// TIA Portal V18 export
// export: Created 2026-06-08T14:19:27.3294129Z, ExportSetting WithDefaults, DisplayName Totally Integrated Automation Portal, DisplayVersion V18, DisplayName TIA Portal Openness, DisplayVersion V18, DisplayName TIA Portal Version Control Interface, DisplayVersion V18, DisplayName STEP 7 Professional, DisplayVersion V18, DisplayName STEP 7 Safety, DisplayVersion V18, DisplayName WinCC Professional, DisplayVersion V18
ORGANIZATION_BLOCK "Main"   // OB1, LAD, ProgramCycle
TITLE = "Main Program Sweep (Cycle)"
{ S7_Optimized_Access := 'TRUE' }
VERSION : 0.1
// stored: AutoNumber true, IsIECCheckEnabled false, SetENOAutomatically false
   VAR_INPUT
      Initial_Call : Bool;   // Initial call of this OB
      Remanence : Bool;   // =True, if remanent data are available
   END_VAR
BEGIN

REGION Network 1: PLC1 - Gọi logic khởi tạo recipe mặc định PLC1
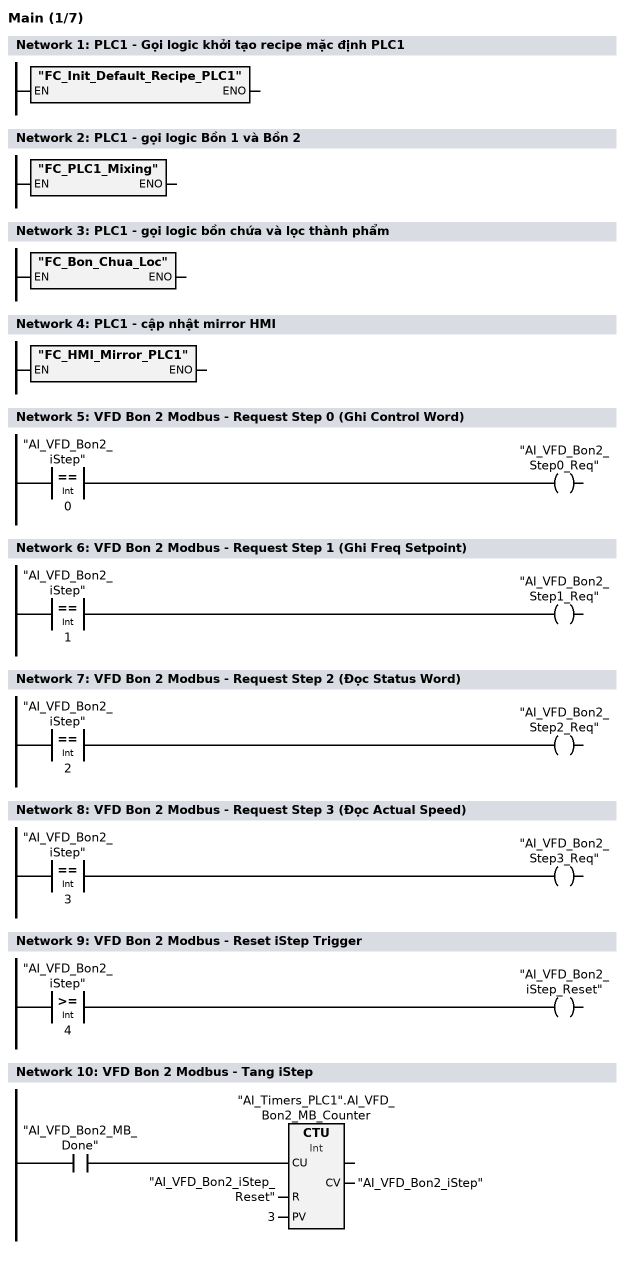
   RUNG wire#powerrail
      "FC_Init_Default_Recipe_PLC1"()
   END_RUNG
   // the same network as SCL:
   "FC_Init_Default_Recipe_PLC1"();
END_REGION

REGION Network 2: PLC1 - gọi logic Bồn 1 và Bồn 2
   RUNG wire#powerrail
      "FC_PLC1_Mixing"()
   END_RUNG
   // the same network as SCL:
   "FC_PLC1_Mixing"();
END_REGION

REGION Network 3: PLC1 - gọi logic bồn chứa và lọc thành phẩm
   RUNG wire#powerrail
      "FC_Bon_Chua_Loc"()
   END_RUNG
   // the same network as SCL:
   "FC_Bon_Chua_Loc"();
END_REGION

REGION Network 4: PLC1 - cập nhật mirror HMI
   RUNG wire#powerrail
      "FC_HMI_Mirror_PLC1"()
   END_RUNG
   // the same network as SCL:
   "FC_HMI_Mirror_PLC1"();
END_REGION

REGION Network 5: VFD Bon 2 Modbus - Request Step 0 (Ghi Control Word)
   RUNG wire#powerrail
      { S7_Templates := "SrcType := Int" } EQ_Contact(in1 := "AI_VFD_Bon2_iStep", in2 := 0)
      Coil( "AI_VFD_Bon2_Step0_Req" )
   END_RUNG
   // the same network as SCL:
   "AI_VFD_Bon2_Step0_Req" := "AI_VFD_Bon2_iStep" = 0;
END_REGION

REGION Network 6: VFD Bon 2 Modbus - Request Step 1 (Ghi Freq Setpoint)
   RUNG wire#powerrail
      { S7_Templates := "SrcType := Int" } EQ_Contact(in1 := "AI_VFD_Bon2_iStep", in2 := 1)
      Coil( "AI_VFD_Bon2_Step1_Req" )
   END_RUNG
   // the same network as SCL:
   "AI_VFD_Bon2_Step1_Req" := "AI_VFD_Bon2_iStep" = 1;
END_REGION

REGION Network 7: VFD Bon 2 Modbus - Request Step 2 (Đọc Status Word)
   RUNG wire#powerrail
      { S7_Templates := "SrcType := Int" } EQ_Contact(in1 := "AI_VFD_Bon2_iStep", in2 := 2)
      Coil( "AI_VFD_Bon2_Step2_Req" )
   END_RUNG
   // the same network as SCL:
   "AI_VFD_Bon2_Step2_Req" := "AI_VFD_Bon2_iStep" = 2;
END_REGION

REGION Network 8: VFD Bon 2 Modbus - Request Step 3 (Đọc Actual Speed)
   RUNG wire#powerrail
      { S7_Templates := "SrcType := Int" } EQ_Contact(in1 := "AI_VFD_Bon2_iStep", in2 := 3)
      Coil( "AI_VFD_Bon2_Step3_Req" )
   END_RUNG
   // the same network as SCL:
   "AI_VFD_Bon2_Step3_Req" := "AI_VFD_Bon2_iStep" = 3;
END_REGION

REGION Network 9: VFD Bon 2 Modbus - Reset iStep Trigger
   RUNG wire#powerrail
      { S7_Templates := "SrcType := Int" } GE_Contact(in1 := "AI_VFD_Bon2_iStep", in2 := 4)
      Coil( "AI_VFD_Bon2_iStep_Reset" )
   END_RUNG
   // the same network as SCL:
   "AI_VFD_Bon2_iStep_Reset" := "AI_VFD_Bon2_iStep" >= 4;
END_REGION

REGION Network 10: VFD Bon 2 Modbus - Tang iStep
   RUNG wire#powerrail
      Contact( "AI_VFD_Bon2_MB_Done" )
      { S7_Templates := "value_type := Int" } "AI_Timers_PLC1".AI_VFD_Bon2_MB_Counter.CTU(r := "AI_VFD_Bon2_iStep_Reset", pv := 3, cv => "AI_VFD_Bon2_iStep")
   END_RUNG
   // the same network as SCL:
   "AI_Timers_PLC1".AI_VFD_Bon2_MB_Counter.CTU(CU := "AI_VFD_Bon2_MB_Done",
                           R := "AI_VFD_Bon2_iStep_Reset",
                           PV := 3,
                           CV => "AI_VFD_Bon2_iStep");
END_REGION

REGION Network 11: VFD Bon 2 Modbus - Khoi tao RS-485
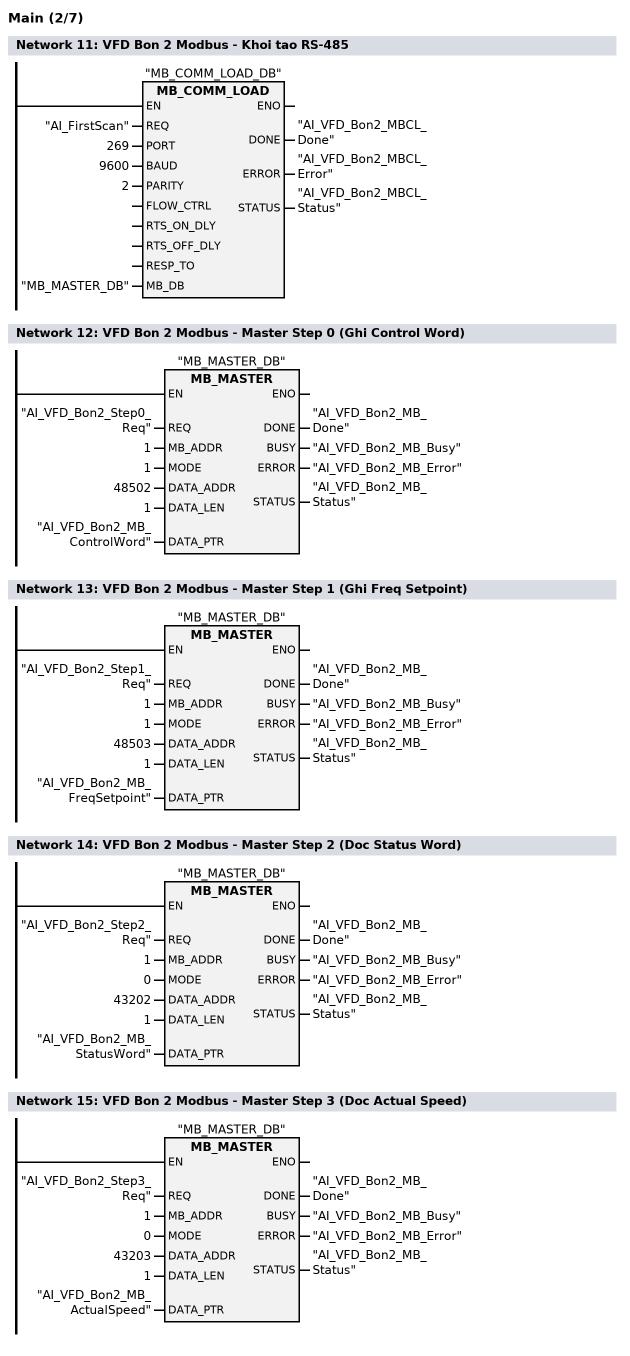
   RUNG wire#powerrail
      "MB_COMM_LOAD_DB".MB_COMM_LOAD(REQ := "AI_FirstScan", PORT := 269, BAUD := 9600, PARITY := 2, FLOW_CTRL :=, RTS_ON_DLY :=, RTS_OFF_DLY :=, RESP_TO :=, MB_DB := "MB_MASTER_DB", DONE => "AI_VFD_Bon2_MBCL_Done", ERROR => "AI_VFD_Bon2_MBCL_Error", STATUS => "AI_VFD_Bon2_MBCL_Status")
   END_RUNG
   // the same network as SCL:
   "MB_COMM_LOAD_DB"(REQ := "AI_FirstScan",   // MB_COMM_LOAD
                     PORT := 269,
                     BAUD := 9600,
                     PARITY := 2,
                     MB_DB := "MB_MASTER_DB",
                     DONE => "AI_VFD_Bon2_MBCL_Done",
                     ERROR => "AI_VFD_Bon2_MBCL_Error",
                     STATUS => "AI_VFD_Bon2_MBCL_Status");
END_REGION

REGION Network 12: VFD Bon 2 Modbus - Master Step 0 (Ghi Control Word)
   RUNG wire#powerrail
      "MB_MASTER_DB".MB_MASTER(REQ := "AI_VFD_Bon2_Step0_Req", MB_ADDR := 1, MODE := 1, DATA_ADDR := 48502, DATA_LEN := 1, DATA_PTR := "AI_VFD_Bon2_MB_ControlWord", DONE => "AI_VFD_Bon2_MB_Done", BUSY => "AI_VFD_Bon2_MB_Busy", ERROR => "AI_VFD_Bon2_MB_Error", STATUS => "AI_VFD_Bon2_MB_Status")
   END_RUNG
   // the same network as SCL:
   "MB_MASTER_DB"(REQ := "AI_VFD_Bon2_Step0_Req",   // MB_MASTER
                  MB_ADDR := 1,
                  MODE := 1,
                  DATA_ADDR := 48502,
                  DATA_LEN := 1,
                  DATA_PTR := "AI_VFD_Bon2_MB_ControlWord",
                  DONE => "AI_VFD_Bon2_MB_Done",
                  BUSY => "AI_VFD_Bon2_MB_Busy",
                  ERROR => "AI_VFD_Bon2_MB_Error",
                  STATUS => "AI_VFD_Bon2_MB_Status");
END_REGION

REGION Network 13: VFD Bon 2 Modbus - Master Step 1 (Ghi Freq Setpoint)
   RUNG wire#powerrail
      "MB_MASTER_DB".MB_MASTER(REQ := "AI_VFD_Bon2_Step1_Req", MB_ADDR := 1, MODE := 1, DATA_ADDR := 48503, DATA_LEN := 1, DATA_PTR := "AI_VFD_Bon2_MB_FreqSetpoint", DONE => "AI_VFD_Bon2_MB_Done", BUSY => "AI_VFD_Bon2_MB_Busy", ERROR => "AI_VFD_Bon2_MB_Error", STATUS => "AI_VFD_Bon2_MB_Status")
   END_RUNG
   // the same network as SCL:
   "MB_MASTER_DB"(REQ := "AI_VFD_Bon2_Step1_Req",   // MB_MASTER
                  MB_ADDR := 1,
                  MODE := 1,
                  DATA_ADDR := 48503,
                  DATA_LEN := 1,
                  DATA_PTR := "AI_VFD_Bon2_MB_FreqSetpoint",
                  DONE => "AI_VFD_Bon2_MB_Done",
                  BUSY => "AI_VFD_Bon2_MB_Busy",
                  ERROR => "AI_VFD_Bon2_MB_Error",
                  STATUS => "AI_VFD_Bon2_MB_Status");
END_REGION

REGION Network 14: VFD Bon 2 Modbus - Master Step 2 (Doc Status Word)
   RUNG wire#powerrail
      "MB_MASTER_DB".MB_MASTER(REQ := "AI_VFD_Bon2_Step2_Req", MB_ADDR := 1, MODE := 0, DATA_ADDR := 43202, DATA_LEN := 1, DATA_PTR := "AI_VFD_Bon2_MB_StatusWord", DONE => "AI_VFD_Bon2_MB_Done", BUSY => "AI_VFD_Bon2_MB_Busy", ERROR => "AI_VFD_Bon2_MB_Error", STATUS => "AI_VFD_Bon2_MB_Status")
   END_RUNG
   // the same network as SCL:
   "MB_MASTER_DB"(REQ := "AI_VFD_Bon2_Step2_Req",   // MB_MASTER
                  MB_ADDR := 1,
                  MODE := 0,
                  DATA_ADDR := 43202,
                  DATA_LEN := 1,
                  DATA_PTR := "AI_VFD_Bon2_MB_StatusWord",
                  DONE => "AI_VFD_Bon2_MB_Done",
                  BUSY => "AI_VFD_Bon2_MB_Busy",
                  ERROR => "AI_VFD_Bon2_MB_Error",
                  STATUS => "AI_VFD_Bon2_MB_Status");
END_REGION

REGION Network 15: VFD Bon 2 Modbus - Master Step 3 (Doc Actual Speed)
   RUNG wire#powerrail
      "MB_MASTER_DB".MB_MASTER(REQ := "AI_VFD_Bon2_Step3_Req", MB_ADDR := 1, MODE := 0, DATA_ADDR := 43203, DATA_LEN := 1, DATA_PTR := "AI_VFD_Bon2_MB_ActualSpeed", DONE => "AI_VFD_Bon2_MB_Done", BUSY => "AI_VFD_Bon2_MB_Busy", ERROR => "AI_VFD_Bon2_MB_Error", STATUS => "AI_VFD_Bon2_MB_Status")
   END_RUNG
   // the same network as SCL:
   "MB_MASTER_DB"(REQ := "AI_VFD_Bon2_Step3_Req",   // MB_MASTER
                  MB_ADDR := 1,
                  MODE := 0,
                  DATA_ADDR := 43203,
                  DATA_LEN := 1,
                  DATA_PTR := "AI_VFD_Bon2_MB_ActualSpeed",
                  DONE => "AI_VFD_Bon2_MB_Done",
                  BUSY => "AI_VFD_Bon2_MB_Busy",
                  ERROR => "AI_VFD_Bon2_MB_Error",
                  STATUS => "AI_VFD_Bon2_MB_Status");
END_REGION

REGION Network 16: Handshake Client - Reset Any Cmd Edge Flag
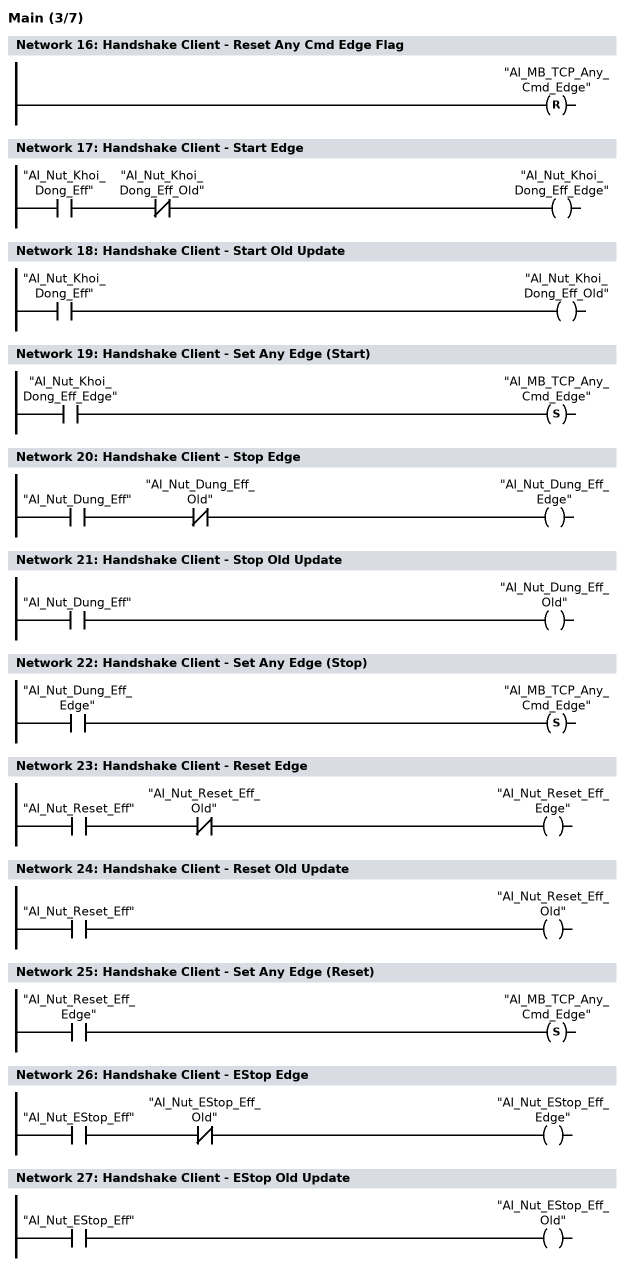
   RUNG wire#powerrail
      R_Coil( "AI_MB_TCP_Any_Cmd_Edge" )
   END_RUNG
   // the same network as SCL:
   "AI_MB_TCP_Any_Cmd_Edge" := FALSE;
END_REGION

REGION Network 17: Handshake Client - Start Edge
   RUNG wire#powerrail
      Contact( "AI_Nut_Khoi_Dong_Eff" )
      I_Contact( "AI_Nut_Khoi_Dong_Eff_Old" )
      Coil( "AI_Nut_Khoi_Dong_Eff_Edge" )
   END_RUNG
   // the same network as SCL:
   "AI_Nut_Khoi_Dong_Eff_Edge" := "AI_Nut_Khoi_Dong_Eff" AND NOT "AI_Nut_Khoi_Dong_Eff_Old";
END_REGION

REGION Network 18: Handshake Client - Start Old Update
   RUNG wire#powerrail
      Contact( "AI_Nut_Khoi_Dong_Eff" )
      Coil( "AI_Nut_Khoi_Dong_Eff_Old" )
   END_RUNG
   // the same network as SCL:
   "AI_Nut_Khoi_Dong_Eff_Old" := "AI_Nut_Khoi_Dong_Eff";
END_REGION

REGION Network 19: Handshake Client - Set Any Edge (Start)
   RUNG wire#powerrail
      Contact( "AI_Nut_Khoi_Dong_Eff_Edge" )
      S_Coil( "AI_MB_TCP_Any_Cmd_Edge" )
   END_RUNG
   // the same network as SCL:
   IF "AI_Nut_Khoi_Dong_Eff_Edge" THEN "AI_MB_TCP_Any_Cmd_Edge" := TRUE; END_IF;
END_REGION

REGION Network 20: Handshake Client - Stop Edge
   RUNG wire#powerrail
      Contact( "AI_Nut_Dung_Eff" )
      I_Contact( "AI_Nut_Dung_Eff_Old" )
      Coil( "AI_Nut_Dung_Eff_Edge" )
   END_RUNG
   // the same network as SCL:
   "AI_Nut_Dung_Eff_Edge" := "AI_Nut_Dung_Eff" AND NOT "AI_Nut_Dung_Eff_Old";
END_REGION

REGION Network 21: Handshake Client - Stop Old Update
   RUNG wire#powerrail
      Contact( "AI_Nut_Dung_Eff" )
      Coil( "AI_Nut_Dung_Eff_Old" )
   END_RUNG
   // the same network as SCL:
   "AI_Nut_Dung_Eff_Old" := "AI_Nut_Dung_Eff";
END_REGION

REGION Network 22: Handshake Client - Set Any Edge (Stop)
   RUNG wire#powerrail
      Contact( "AI_Nut_Dung_Eff_Edge" )
      S_Coil( "AI_MB_TCP_Any_Cmd_Edge" )
   END_RUNG
   // the same network as SCL:
   IF "AI_Nut_Dung_Eff_Edge" THEN "AI_MB_TCP_Any_Cmd_Edge" := TRUE; END_IF;
END_REGION

REGION Network 23: Handshake Client - Reset Edge
   RUNG wire#powerrail
      Contact( "AI_Nut_Reset_Eff" )
      I_Contact( "AI_Nut_Reset_Eff_Old" )
      Coil( "AI_Nut_Reset_Eff_Edge" )
   END_RUNG
   // the same network as SCL:
   "AI_Nut_Reset_Eff_Edge" := "AI_Nut_Reset_Eff" AND NOT "AI_Nut_Reset_Eff_Old";
END_REGION

REGION Network 24: Handshake Client - Reset Old Update
   RUNG wire#powerrail
      Contact( "AI_Nut_Reset_Eff" )
      Coil( "AI_Nut_Reset_Eff_Old" )
   END_RUNG
   // the same network as SCL:
   "AI_Nut_Reset_Eff_Old" := "AI_Nut_Reset_Eff";
END_REGION

REGION Network 25: Handshake Client - Set Any Edge (Reset)
   RUNG wire#powerrail
      Contact( "AI_Nut_Reset_Eff_Edge" )
      S_Coil( "AI_MB_TCP_Any_Cmd_Edge" )
   END_RUNG
   // the same network as SCL:
   IF "AI_Nut_Reset_Eff_Edge" THEN "AI_MB_TCP_Any_Cmd_Edge" := TRUE; END_IF;
END_REGION

REGION Network 26: Handshake Client - EStop Edge
   RUNG wire#powerrail
      Contact( "AI_Nut_EStop_Eff" )
      I_Contact( "AI_Nut_EStop_Eff_Old" )
      Coil( "AI_Nut_EStop_Eff_Edge" )
   END_RUNG
   // the same network as SCL:
   "AI_Nut_EStop_Eff_Edge" := "AI_Nut_EStop_Eff" AND NOT "AI_Nut_EStop_Eff_Old";
END_REGION

REGION Network 27: Handshake Client - EStop Old Update
   RUNG wire#powerrail
      Contact( "AI_Nut_EStop_Eff" )
      Coil( "AI_Nut_EStop_Eff_Old" )
   END_RUNG
   // the same network as SCL:
   "AI_Nut_EStop_Eff_Old" := "AI_Nut_EStop_Eff";
END_REGION

REGION Network 28: Handshake Client - Set Any Edge (EStop)
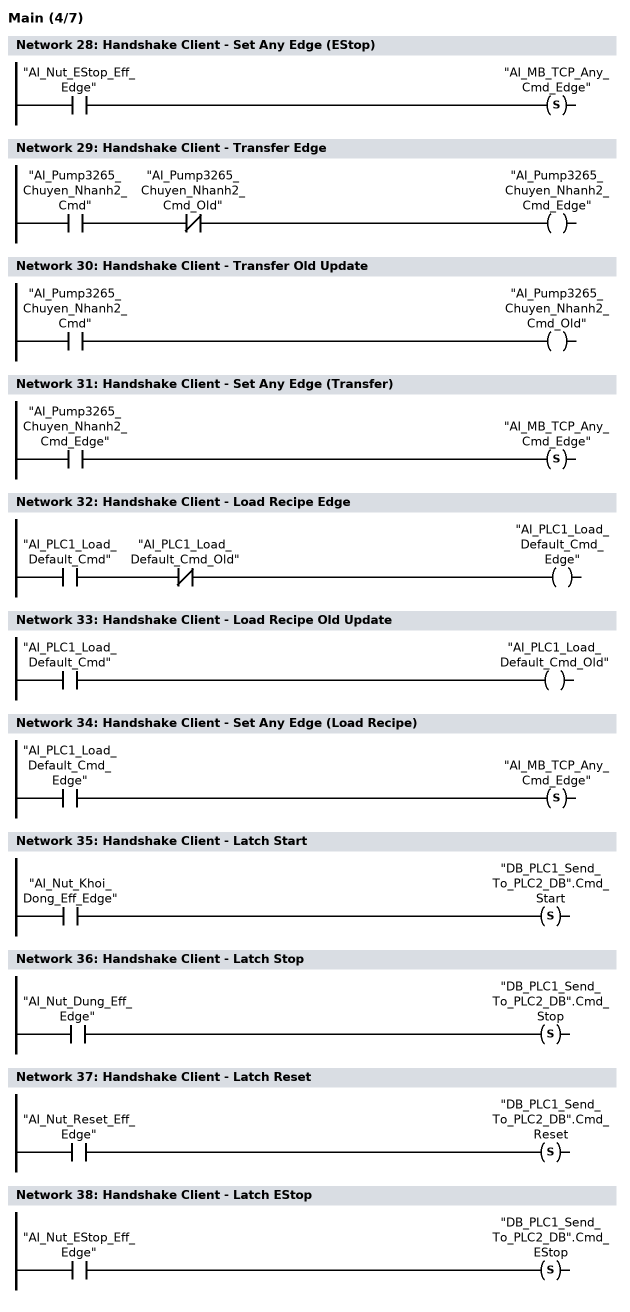
   RUNG wire#powerrail
      Contact( "AI_Nut_EStop_Eff_Edge" )
      S_Coil( "AI_MB_TCP_Any_Cmd_Edge" )
   END_RUNG
   // the same network as SCL:
   IF "AI_Nut_EStop_Eff_Edge" THEN "AI_MB_TCP_Any_Cmd_Edge" := TRUE; END_IF;
END_REGION

REGION Network 29: Handshake Client - Transfer Edge
   RUNG wire#powerrail
      Contact( "AI_Pump3265_Chuyen_Nhanh2_Cmd" )
      I_Contact( "AI_Pump3265_Chuyen_Nhanh2_Cmd_Old" )
      Coil( "AI_Pump3265_Chuyen_Nhanh2_Cmd_Edge" )
   END_RUNG
   // the same network as SCL:
   "AI_Pump3265_Chuyen_Nhanh2_Cmd_Edge" := "AI_Pump3265_Chuyen_Nhanh2_Cmd" AND NOT "AI_Pump3265_Chuyen_Nhanh2_Cmd_Old";
END_REGION

REGION Network 30: Handshake Client - Transfer Old Update
   RUNG wire#powerrail
      Contact( "AI_Pump3265_Chuyen_Nhanh2_Cmd" )
      Coil( "AI_Pump3265_Chuyen_Nhanh2_Cmd_Old" )
   END_RUNG
   // the same network as SCL:
   "AI_Pump3265_Chuyen_Nhanh2_Cmd_Old" := "AI_Pump3265_Chuyen_Nhanh2_Cmd";
END_REGION

REGION Network 31: Handshake Client - Set Any Edge (Transfer)
   RUNG wire#powerrail
      Contact( "AI_Pump3265_Chuyen_Nhanh2_Cmd_Edge" )
      S_Coil( "AI_MB_TCP_Any_Cmd_Edge" )
   END_RUNG
   // the same network as SCL:
   IF "AI_Pump3265_Chuyen_Nhanh2_Cmd_Edge" THEN "AI_MB_TCP_Any_Cmd_Edge" := TRUE; END_IF;
END_REGION

REGION Network 32: Handshake Client - Load Recipe Edge
   RUNG wire#powerrail
      Contact( "AI_PLC1_Load_Default_Cmd" )
      I_Contact( "AI_PLC1_Load_Default_Cmd_Old" )
      Coil( "AI_PLC1_Load_Default_Cmd_Edge" )
   END_RUNG
   // the same network as SCL:
   "AI_PLC1_Load_Default_Cmd_Edge" := "AI_PLC1_Load_Default_Cmd" AND NOT "AI_PLC1_Load_Default_Cmd_Old";
END_REGION

REGION Network 33: Handshake Client - Load Recipe Old Update
   RUNG wire#powerrail
      Contact( "AI_PLC1_Load_Default_Cmd" )
      Coil( "AI_PLC1_Load_Default_Cmd_Old" )
   END_RUNG
   // the same network as SCL:
   "AI_PLC1_Load_Default_Cmd_Old" := "AI_PLC1_Load_Default_Cmd";
END_REGION

REGION Network 34: Handshake Client - Set Any Edge (Load Recipe)
   RUNG wire#powerrail
      Contact( "AI_PLC1_Load_Default_Cmd_Edge" )
      S_Coil( "AI_MB_TCP_Any_Cmd_Edge" )
   END_RUNG
   // the same network as SCL:
   IF "AI_PLC1_Load_Default_Cmd_Edge" THEN "AI_MB_TCP_Any_Cmd_Edge" := TRUE; END_IF;
END_REGION

REGION Network 35: Handshake Client - Latch Start
   RUNG wire#powerrail
      Contact( "AI_Nut_Khoi_Dong_Eff_Edge" )
      S_Coil( "DB_PLC1_Send_To_PLC2_DB".Cmd_Start )
   END_RUNG
   // the same network as SCL:
   IF "AI_Nut_Khoi_Dong_Eff_Edge" THEN "DB_PLC1_Send_To_PLC2_DB".Cmd_Start := TRUE; END_IF;
END_REGION

REGION Network 36: Handshake Client - Latch Stop
   RUNG wire#powerrail
      Contact( "AI_Nut_Dung_Eff_Edge" )
      S_Coil( "DB_PLC1_Send_To_PLC2_DB".Cmd_Stop )
   END_RUNG
   // the same network as SCL:
   IF "AI_Nut_Dung_Eff_Edge" THEN "DB_PLC1_Send_To_PLC2_DB".Cmd_Stop := TRUE; END_IF;
END_REGION

REGION Network 37: Handshake Client - Latch Reset
   RUNG wire#powerrail
      Contact( "AI_Nut_Reset_Eff_Edge" )
      S_Coil( "DB_PLC1_Send_To_PLC2_DB".Cmd_Reset )
   END_RUNG
   // the same network as SCL:
   IF "AI_Nut_Reset_Eff_Edge" THEN "DB_PLC1_Send_To_PLC2_DB".Cmd_Reset := TRUE; END_IF;
END_REGION

REGION Network 38: Handshake Client - Latch EStop
   RUNG wire#powerrail
      Contact( "AI_Nut_EStop_Eff_Edge" )
      S_Coil( "DB_PLC1_Send_To_PLC2_DB".Cmd_EStop )
   END_RUNG
   // the same network as SCL:
   IF "AI_Nut_EStop_Eff_Edge" THEN "DB_PLC1_Send_To_PLC2_DB".Cmd_EStop := TRUE; END_IF;
END_REGION

REGION Network 39: Handshake Client - Latch Transfer
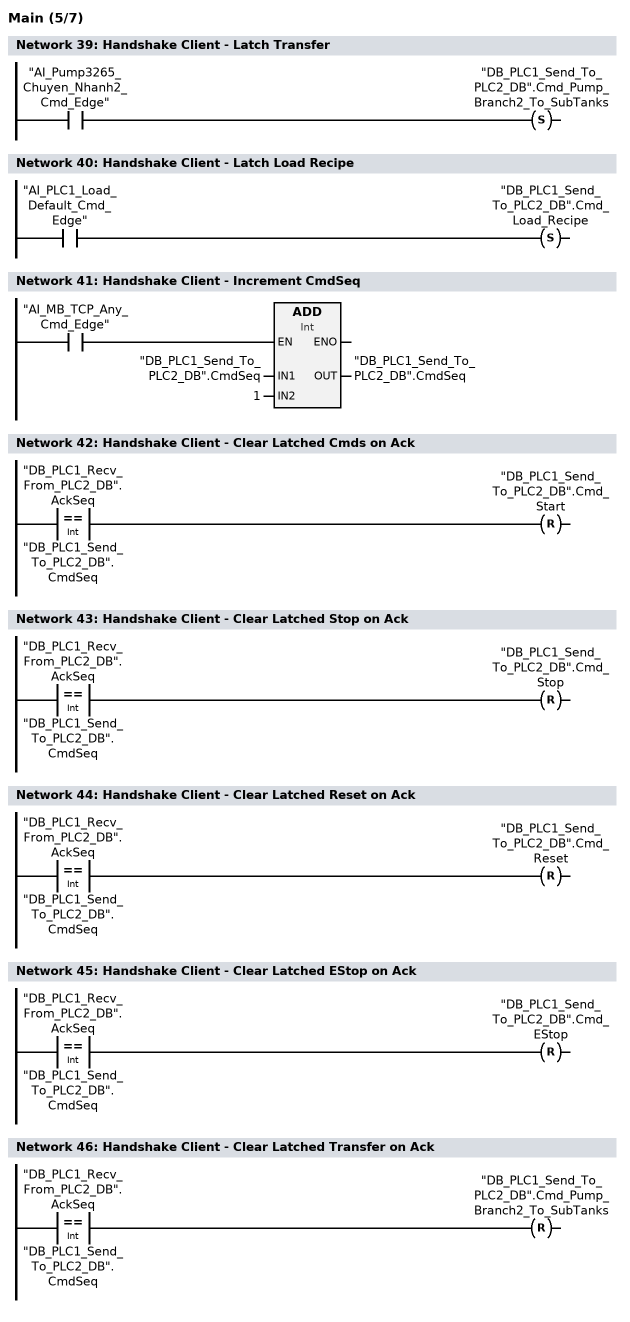
   RUNG wire#powerrail
      Contact( "AI_Pump3265_Chuyen_Nhanh2_Cmd_Edge" )
      S_Coil( "DB_PLC1_Send_To_PLC2_DB".Cmd_Pump_Branch2_To_SubTanks )
   END_RUNG
   // the same network as SCL:
   IF "AI_Pump3265_Chuyen_Nhanh2_Cmd_Edge" THEN
       "DB_PLC1_Send_To_PLC2_DB".Cmd_Pump_Branch2_To_SubTanks := TRUE;
   END_IF;
END_REGION

REGION Network 40: Handshake Client - Latch Load Recipe
   RUNG wire#powerrail
      Contact( "AI_PLC1_Load_Default_Cmd_Edge" )
      S_Coil( "DB_PLC1_Send_To_PLC2_DB".Cmd_Load_Recipe )
   END_RUNG
   // the same network as SCL:
   IF "AI_PLC1_Load_Default_Cmd_Edge" THEN "DB_PLC1_Send_To_PLC2_DB".Cmd_Load_Recipe := TRUE; END_IF;
END_REGION

REGION Network 41: Handshake Client - Increment CmdSeq
   RUNG wire#powerrail
      Contact( "AI_MB_TCP_Any_Cmd_Edge" )
      { S7_Templates := "SrcType := Int"; S7_GenerateENO := "TRUE" } Add(in1 := "DB_PLC1_Send_To_PLC2_DB".CmdSeq, in2 := 1, out => "DB_PLC1_Send_To_PLC2_DB".CmdSeq)
   END_RUNG
   // the same network as SCL:
   IF "AI_MB_TCP_Any_Cmd_Edge" THEN
       "DB_PLC1_Send_To_PLC2_DB".CmdSeq := "DB_PLC1_Send_To_PLC2_DB".CmdSeq + 1;
   END_IF;
END_REGION

REGION Network 42: Handshake Client - Clear Latched Cmds on Ack
   RUNG wire#powerrail
      { S7_Templates := "SrcType := Int" } EQ_Contact(in1 := "DB_PLC1_Recv_From_PLC2_DB".AckSeq, in2 := "DB_PLC1_Send_To_PLC2_DB".CmdSeq)
      R_Coil( "DB_PLC1_Send_To_PLC2_DB".Cmd_Start )
   END_RUNG
   // the same network as SCL:
   IF "DB_PLC1_Recv_From_PLC2_DB".AckSeq = "DB_PLC1_Send_To_PLC2_DB".CmdSeq THEN
       "DB_PLC1_Send_To_PLC2_DB".Cmd_Start := FALSE;
   END_IF;
END_REGION

REGION Network 43: Handshake Client - Clear Latched Stop on Ack
   RUNG wire#powerrail
      { S7_Templates := "SrcType := Int" } EQ_Contact(in1 := "DB_PLC1_Recv_From_PLC2_DB".AckSeq, in2 := "DB_PLC1_Send_To_PLC2_DB".CmdSeq)
      R_Coil( "DB_PLC1_Send_To_PLC2_DB".Cmd_Stop )
   END_RUNG
   // the same network as SCL:
   IF "DB_PLC1_Recv_From_PLC2_DB".AckSeq = "DB_PLC1_Send_To_PLC2_DB".CmdSeq THEN
       "DB_PLC1_Send_To_PLC2_DB".Cmd_Stop := FALSE;
   END_IF;
END_REGION

REGION Network 44: Handshake Client - Clear Latched Reset on Ack
   RUNG wire#powerrail
      { S7_Templates := "SrcType := Int" } EQ_Contact(in1 := "DB_PLC1_Recv_From_PLC2_DB".AckSeq, in2 := "DB_PLC1_Send_To_PLC2_DB".CmdSeq)
      R_Coil( "DB_PLC1_Send_To_PLC2_DB".Cmd_Reset )
   END_RUNG
   // the same network as SCL:
   IF "DB_PLC1_Recv_From_PLC2_DB".AckSeq = "DB_PLC1_Send_To_PLC2_DB".CmdSeq THEN
       "DB_PLC1_Send_To_PLC2_DB".Cmd_Reset := FALSE;
   END_IF;
END_REGION

REGION Network 45: Handshake Client - Clear Latched EStop on Ack
   RUNG wire#powerrail
      { S7_Templates := "SrcType := Int" } EQ_Contact(in1 := "DB_PLC1_Recv_From_PLC2_DB".AckSeq, in2 := "DB_PLC1_Send_To_PLC2_DB".CmdSeq)
      R_Coil( "DB_PLC1_Send_To_PLC2_DB".Cmd_EStop )
   END_RUNG
   // the same network as SCL:
   IF "DB_PLC1_Recv_From_PLC2_DB".AckSeq = "DB_PLC1_Send_To_PLC2_DB".CmdSeq THEN
       "DB_PLC1_Send_To_PLC2_DB".Cmd_EStop := FALSE;
   END_IF;
END_REGION

REGION Network 46: Handshake Client - Clear Latched Transfer on Ack
   RUNG wire#powerrail
      { S7_Templates := "SrcType := Int" } EQ_Contact(in1 := "DB_PLC1_Recv_From_PLC2_DB".AckSeq, in2 := "DB_PLC1_Send_To_PLC2_DB".CmdSeq)
      R_Coil( "DB_PLC1_Send_To_PLC2_DB".Cmd_Pump_Branch2_To_SubTanks )
   END_RUNG
   // the same network as SCL:
   IF "DB_PLC1_Recv_From_PLC2_DB".AckSeq = "DB_PLC1_Send_To_PLC2_DB".CmdSeq THEN
       "DB_PLC1_Send_To_PLC2_DB".Cmd_Pump_Branch2_To_SubTanks := FALSE;
   END_IF;
END_REGION

REGION Network 47: Handshake Client - Clear Latched Load Recipe on Ack
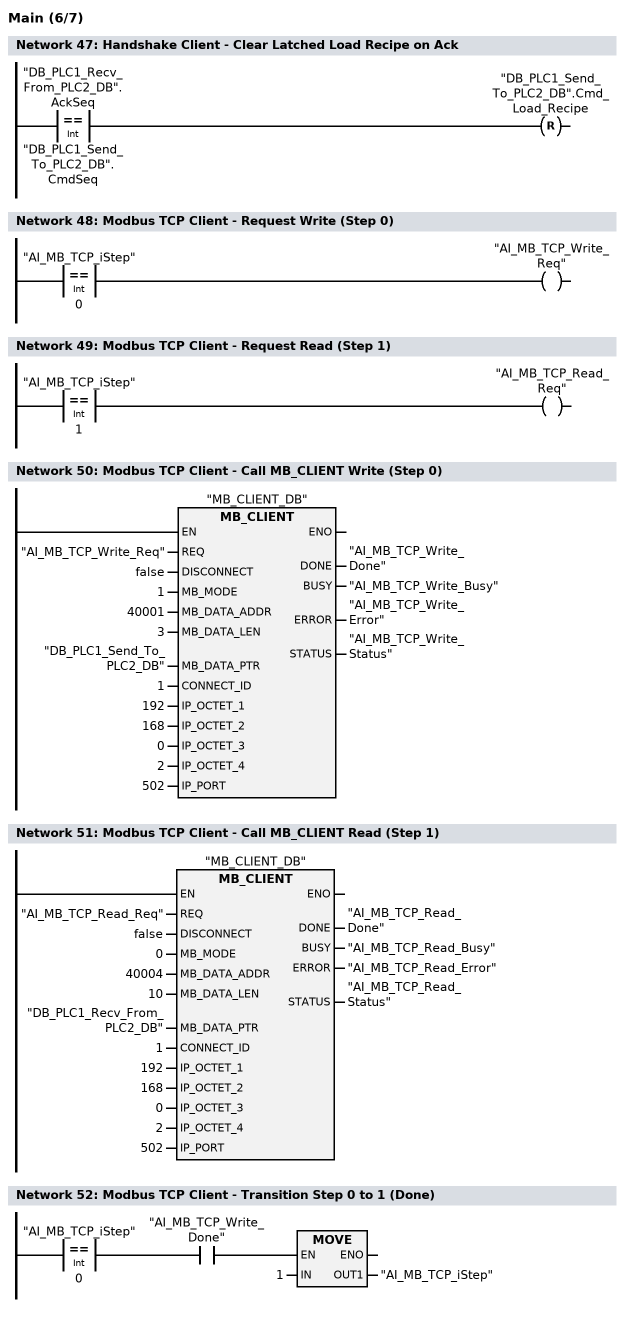
   RUNG wire#powerrail
      { S7_Templates := "SrcType := Int" } EQ_Contact(in1 := "DB_PLC1_Recv_From_PLC2_DB".AckSeq, in2 := "DB_PLC1_Send_To_PLC2_DB".CmdSeq)
      R_Coil( "DB_PLC1_Send_To_PLC2_DB".Cmd_Load_Recipe )
   END_RUNG
   // the same network as SCL:
   IF "DB_PLC1_Recv_From_PLC2_DB".AckSeq = "DB_PLC1_Send_To_PLC2_DB".CmdSeq THEN
       "DB_PLC1_Send_To_PLC2_DB".Cmd_Load_Recipe := FALSE;
   END_IF;
END_REGION

REGION Network 48: Modbus TCP Client - Request Write (Step 0)
   RUNG wire#powerrail
      { S7_Templates := "SrcType := Int" } EQ_Contact(in1 := "AI_MB_TCP_iStep", in2 := 0)
      Coil( "AI_MB_TCP_Write_Req" )
   END_RUNG
   // the same network as SCL:
   "AI_MB_TCP_Write_Req" := "AI_MB_TCP_iStep" = 0;
END_REGION

REGION Network 49: Modbus TCP Client - Request Read (Step 1)
   RUNG wire#powerrail
      { S7_Templates := "SrcType := Int" } EQ_Contact(in1 := "AI_MB_TCP_iStep", in2 := 1)
      Coil( "AI_MB_TCP_Read_Req" )
   END_RUNG
   // the same network as SCL:
   "AI_MB_TCP_Read_Req" := "AI_MB_TCP_iStep" = 1;
END_REGION

REGION Network 50: Modbus TCP Client - Call MB_CLIENT Write (Step 0)
   RUNG wire#powerrail
      { S7_Templates := "[card1200 := 1, card1500 := 0]" } "MB_CLIENT_DB".MB_CLIENT(REQ := "AI_MB_TCP_Write_Req", DISCONNECT := false, MB_MODE := 1, MB_DATA_ADDR := 40001, MB_DATA_LEN := 3, MB_DATA_PTR := "DB_PLC1_Send_To_PLC2_DB", CONNECT_ID := 1, IP_OCTET_1 := 192, IP_OCTET_2 := 168, IP_OCTET_3 := 0, IP_OCTET_4 := 2, IP_PORT := 502, DONE => "AI_MB_TCP_Write_Done", BUSY => "AI_MB_TCP_Write_Busy", ERROR => "AI_MB_TCP_Write_Error", STATUS => "AI_MB_TCP_Write_Status")
   END_RUNG
   // the same network as SCL:
   "MB_CLIENT_DB"(REQ := "AI_MB_TCP_Write_Req",   // MB_CLIENT
                  DISCONNECT := false,
                  MB_MODE := 1,
                  MB_DATA_ADDR := 40001,
                  MB_DATA_LEN := 3,
                  MB_DATA_PTR := "DB_PLC1_Send_To_PLC2_DB",
                  CONNECT_ID := 1,
                  IP_OCTET_1 := 192,
                  IP_OCTET_2 := 168,
                  IP_OCTET_3 := 0,
                  IP_OCTET_4 := 2,
                  IP_PORT := 502,
                  DONE => "AI_MB_TCP_Write_Done",
                  BUSY => "AI_MB_TCP_Write_Busy",
                  ERROR => "AI_MB_TCP_Write_Error",
                  STATUS => "AI_MB_TCP_Write_Status");
END_REGION

REGION Network 51: Modbus TCP Client - Call MB_CLIENT Read (Step 1)
   RUNG wire#powerrail
      { S7_Templates := "[card1200 := 1, card1500 := 0]" } "MB_CLIENT_DB".MB_CLIENT(REQ := "AI_MB_TCP_Read_Req", DISCONNECT := false, MB_MODE := 0, MB_DATA_ADDR := 40004, MB_DATA_LEN := 10, MB_DATA_PTR := "DB_PLC1_Recv_From_PLC2_DB", CONNECT_ID := 1, IP_OCTET_1 := 192, IP_OCTET_2 := 168, IP_OCTET_3 := 0, IP_OCTET_4 := 2, IP_PORT := 502, DONE => "AI_MB_TCP_Read_Done", BUSY => "AI_MB_TCP_Read_Busy", ERROR => "AI_MB_TCP_Read_Error", STATUS => "AI_MB_TCP_Read_Status")
   END_RUNG
   // the same network as SCL:
   "MB_CLIENT_DB"(REQ := "AI_MB_TCP_Read_Req",   // MB_CLIENT
                  DISCONNECT := false,
                  MB_MODE := 0,
                  MB_DATA_ADDR := 40004,
                  MB_DATA_LEN := 10,
                  MB_DATA_PTR := "DB_PLC1_Recv_From_PLC2_DB",
                  CONNECT_ID := 1,
                  IP_OCTET_1 := 192,
                  IP_OCTET_2 := 168,
                  IP_OCTET_3 := 0,
                  IP_OCTET_4 := 2,
                  IP_PORT := 502,
                  DONE => "AI_MB_TCP_Read_Done",
                  BUSY => "AI_MB_TCP_Read_Busy",
                  ERROR => "AI_MB_TCP_Read_Error",
                  STATUS => "AI_MB_TCP_Read_Status");
END_REGION

REGION Network 52: Modbus TCP Client - Transition Step 0 to 1 (Done)
   RUNG wire#powerrail
      { S7_Templates := "SrcType := Int" } EQ_Contact(in1 := "AI_MB_TCP_iStep", in2 := 0)
      Contact( "AI_MB_TCP_Write_Done" )
      { S7_GenerateENO := "TRUE" } Move(in := 1, out1 => "AI_MB_TCP_iStep")
   END_RUNG
   // the same network as SCL:
   IF ("AI_MB_TCP_iStep" = 0) AND "AI_MB_TCP_Write_Done" THEN "AI_MB_TCP_iStep" := 1; END_IF;
END_REGION

REGION Network 53: Modbus TCP Client - Transition Step 0 to 1 (Error)
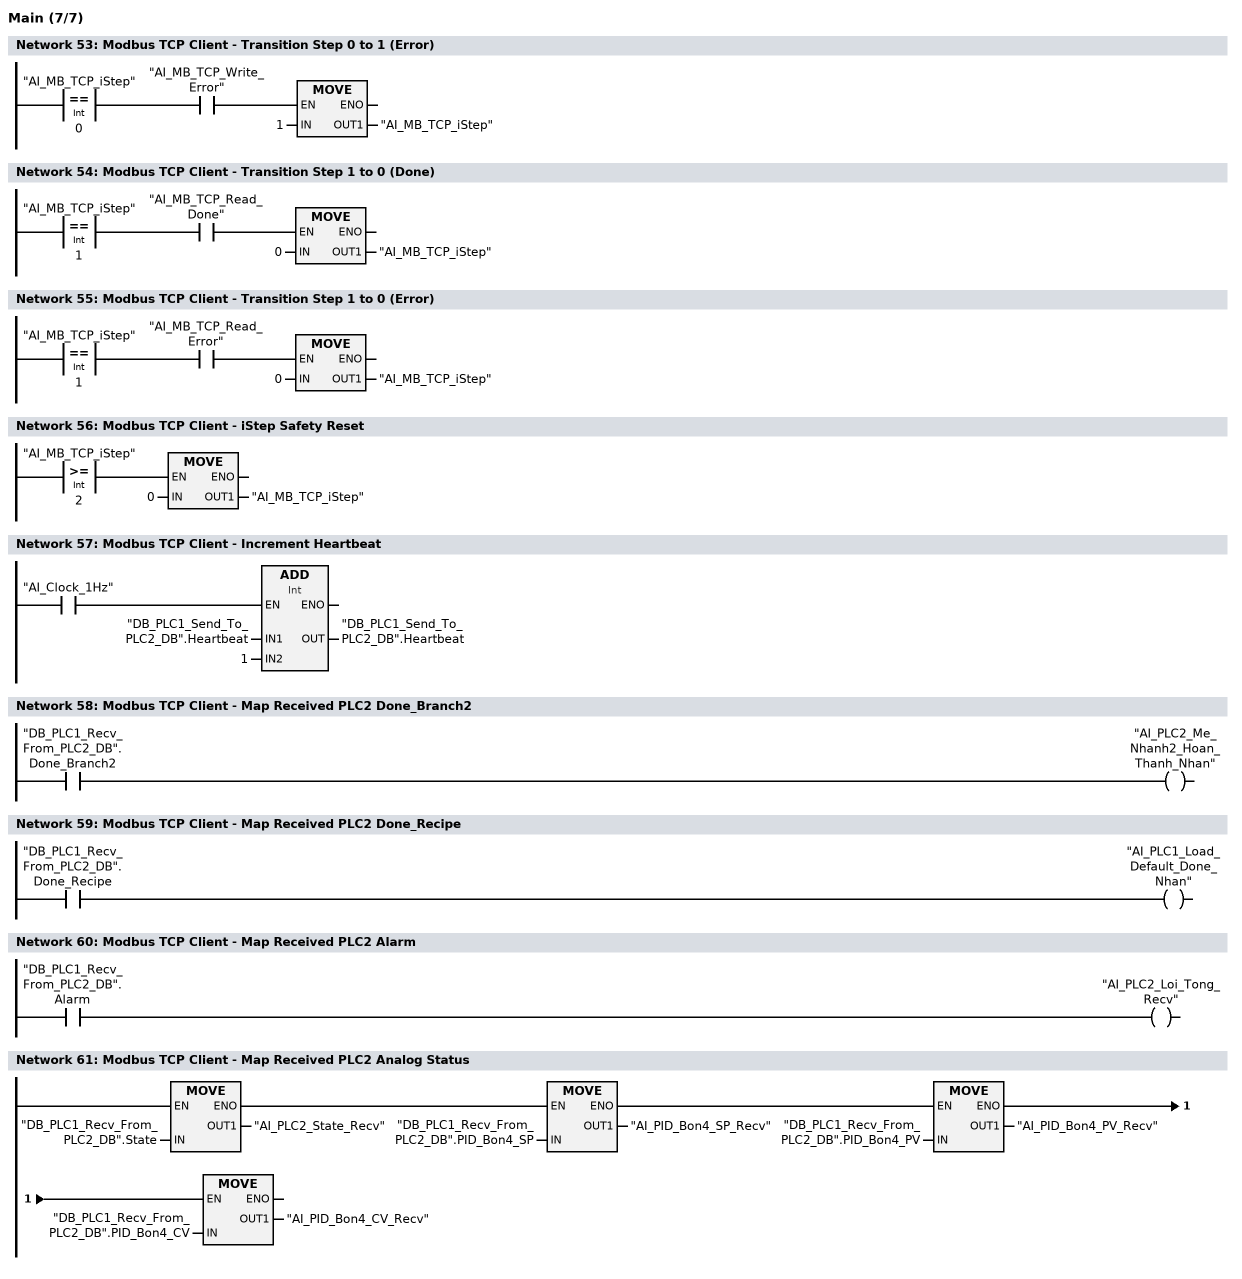
   RUNG wire#powerrail
      { S7_Templates := "SrcType := Int" } EQ_Contact(in1 := "AI_MB_TCP_iStep", in2 := 0)
      Contact( "AI_MB_TCP_Write_Error" )
      { S7_GenerateENO := "TRUE" } Move(in := 1, out1 => "AI_MB_TCP_iStep")
   END_RUNG
   // the same network as SCL:
   IF ("AI_MB_TCP_iStep" = 0) AND "AI_MB_TCP_Write_Error" THEN "AI_MB_TCP_iStep" := 1; END_IF;
END_REGION

REGION Network 54: Modbus TCP Client - Transition Step 1 to 0 (Done)
   RUNG wire#powerrail
      { S7_Templates := "SrcType := Int" } EQ_Contact(in1 := "AI_MB_TCP_iStep", in2 := 1)
      Contact( "AI_MB_TCP_Read_Done" )
      { S7_GenerateENO := "TRUE" } Move(in := 0, out1 => "AI_MB_TCP_iStep")
   END_RUNG
   // the same network as SCL:
   IF ("AI_MB_TCP_iStep" = 1) AND "AI_MB_TCP_Read_Done" THEN "AI_MB_TCP_iStep" := 0; END_IF;
END_REGION

REGION Network 55: Modbus TCP Client - Transition Step 1 to 0 (Error)
   RUNG wire#powerrail
      { S7_Templates := "SrcType := Int" } EQ_Contact(in1 := "AI_MB_TCP_iStep", in2 := 1)
      Contact( "AI_MB_TCP_Read_Error" )
      { S7_GenerateENO := "TRUE" } Move(in := 0, out1 => "AI_MB_TCP_iStep")
   END_RUNG
   // the same network as SCL:
   IF ("AI_MB_TCP_iStep" = 1) AND "AI_MB_TCP_Read_Error" THEN "AI_MB_TCP_iStep" := 0; END_IF;
END_REGION

REGION Network 56: Modbus TCP Client - iStep Safety Reset
   RUNG wire#powerrail
      { S7_Templates := "SrcType := Int" } GE_Contact(in1 := "AI_MB_TCP_iStep", in2 := 2)
      { S7_GenerateENO := "TRUE" } Move(in := 0, out1 => "AI_MB_TCP_iStep")
   END_RUNG
   // the same network as SCL:
   IF "AI_MB_TCP_iStep" >= 2 THEN "AI_MB_TCP_iStep" := 0; END_IF;
END_REGION

REGION Network 57: Modbus TCP Client - Increment Heartbeat
   RUNG wire#powerrail
      Contact( "AI_Clock_1Hz" )
      { S7_Templates := "SrcType := Int"; S7_GenerateENO := "TRUE" } Add(in1 := "DB_PLC1_Send_To_PLC2_DB".Heartbeat, in2 := 1, out => "DB_PLC1_Send_To_PLC2_DB".Heartbeat)
   END_RUNG
   // the same network as SCL:
   IF "AI_Clock_1Hz" THEN
       "DB_PLC1_Send_To_PLC2_DB".Heartbeat := "DB_PLC1_Send_To_PLC2_DB".Heartbeat + 1;
   END_IF;
END_REGION

REGION Network 58: Modbus TCP Client - Map Received PLC2 Done_Branch2
   RUNG wire#powerrail
      Contact( "DB_PLC1_Recv_From_PLC2_DB".Done_Branch2 )
      Coil( "AI_PLC2_Me_Nhanh2_Hoan_Thanh_Nhan" )
   END_RUNG
   // the same network as SCL:
   "AI_PLC2_Me_Nhanh2_Hoan_Thanh_Nhan" := "DB_PLC1_Recv_From_PLC2_DB".Done_Branch2;
END_REGION

REGION Network 59: Modbus TCP Client - Map Received PLC2 Done_Recipe
   RUNG wire#powerrail
      Contact( "DB_PLC1_Recv_From_PLC2_DB".Done_Recipe )
      Coil( "AI_PLC1_Load_Default_Done_Nhan" )
   END_RUNG
   // the same network as SCL:
   "AI_PLC1_Load_Default_Done_Nhan" := "DB_PLC1_Recv_From_PLC2_DB".Done_Recipe;
END_REGION

REGION Network 60: Modbus TCP Client - Map Received PLC2 Alarm
   RUNG wire#powerrail
      Contact( "DB_PLC1_Recv_From_PLC2_DB".Alarm )
      Coil( "AI_PLC2_Loi_Tong_Recv" )
   END_RUNG
   // the same network as SCL:
   "AI_PLC2_Loi_Tong_Recv" := "DB_PLC1_Recv_From_PLC2_DB".Alarm;
END_REGION

REGION Network 61: Modbus TCP Client - Map Received PLC2 Analog Status
   RUNG wire#powerrail
      { S7_GenerateENO := "TRUE" } Move(in := "DB_PLC1_Recv_From_PLC2_DB".State, out1 => "AI_PLC2_State_Recv")
      { S7_GenerateENO := "TRUE" } Move(in := "DB_PLC1_Recv_From_PLC2_DB".PID_Bon4_SP, out1 => "AI_PID_Bon4_SP_Recv")
      { S7_GenerateENO := "TRUE" } Move(in := "DB_PLC1_Recv_From_PLC2_DB".PID_Bon4_PV, out1 => "AI_PID_Bon4_PV_Recv")
      { S7_GenerateENO := "TRUE" } Move(in := "DB_PLC1_Recv_From_PLC2_DB".PID_Bon4_CV, out1 => "AI_PID_Bon4_CV_Recv")
   END_RUNG
   // the same network as SCL:
   // ENO of a box is taken as its EN; it also drops when the box reports an error
   "AI_PLC2_State_Recv" := "DB_PLC1_Recv_From_PLC2_DB".State;
   "AI_PID_Bon4_SP_Recv" := "DB_PLC1_Recv_From_PLC2_DB".PID_Bon4_SP;
   "AI_PID_Bon4_PV_Recv" := "DB_PLC1_Recv_From_PLC2_DB".PID_Bon4_PV;
   "AI_PID_Bon4_CV_Recv" := "DB_PLC1_Recv_From_PLC2_DB".PID_Bon4_CV;
END_REGION
END_ORGANIZATION_BLOCK
